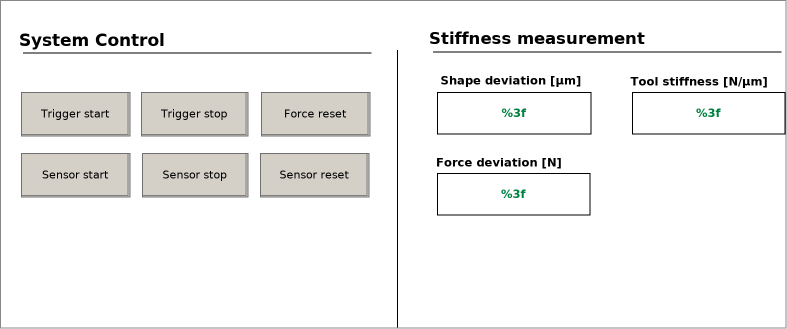
VISUALIZATION VISUALISATION_STIFFNESS_PROCESS  // 787x329
    Button (21,92 109x44), "Trigger start"
        OnMouseClick: execute { VARIABLES.CAN_TRIGGER_STATE:=1; }
    Button (141,92 107x44), "Trigger stop"
        OnMouseClick: execute { VARIABLES.CAN_TRIGGER_STATE:=0; }
    Button (21,153 109x44), "Sensor start"
        OnMouseClick: execute { CAN_CONTROL_STATE:=1; }
    Button (142,153 106x44), "Sensor stop"
        OnMouseClick: execute { CAN_CONTROL_STATE:=0; }
    Button (260,153 109x44), "Sensor reset"
        OnMouseClick: execute { CAN_CONTROL_STATE:=2; }
    Button (261,92 109x44), "Force reset"
        OnMouseClick: execute { VARIABLES.FORCE_RESET:=1; }
    Rectangle (17,25 150x30), "System Control"
    Line (371,53) (23,53)
    Rectangle (428,31 218x15), "Stiffness measurement"
    Rectangle (632,92 153x42), "%3f", text variable: VARIABLES.TOOL_STIFFNESS_SELC_PTS[2,3]
    Rectangle (437,92 154x42), "%3f", text variable: VARIABLES.SHAPE_DEVIATION
    Rectangle (437,173 153x42), "%3f", text variable: VARIABLES.FORCE_DEVIATION[2]
    Rectangle (437,73 148x15), "Shape deviation [µm]"
    Rectangle (437,155 124x15), "Force deviation [N]"
    Rectangle (632,74 135x15), "Tool stiffness [N/µm]"
    Line (397,50) (397,327)
    Line (781,52) (433,52)
END_VISUALIZATION

(* stored: Version 1.1.0.1, ProductVersion 3.1.0.26
   Visu VISUALISATION_STIFFNESS_PROCESS: Id {284a3e38-6bb2-4737-813d-06a8721fd8af} *)
